FUNCTION_BLOCK ConvRobCtrl (* Basic Function Block Type *)
  (* Standard: 61499-2 *)
  (* Version 0.0, 5/12/2018, Aalto_IT, nxtControl GmbH, Template *)
  PACKAGE Main;
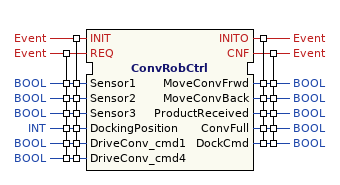
  EVENT_INPUT
    INIT WITH Sensor1, Sensor2, Sensor3, DockingPosition, DriveConv_cmd1, DriveConv_cmd4; (* Initialization Request *)
    REQ WITH Sensor1, Sensor2, Sensor3, DockingPosition, DriveConv_cmd1, DriveConv_cmd4; (* Normal Execution Request *)
  END_EVENT
  EVENT_OUTPUT
    INITO WITH MoveConvFrwd, MoveConvBack, ProductReceived, ConvFull, DockCmd; (* Initialization Confirm *)
    CNF WITH MoveConvFrwd, MoveConvBack, ProductReceived, ConvFull, DockCmd; (* Execution Confirmation *)
  END_EVENT
  VAR_INPUT
    Sensor1 : BOOL; (* Input event qualifier *)
    Sensor2 : BOOL;
    Sensor3 : BOOL;
    DockingPosition : INT;
    DriveConv_cmd1 : BOOL;
    DriveConv_cmd4 : BOOL;
  END_VAR
  VAR_OUTPUT
    MoveConvFrwd : BOOL; (* Output event qualifier *)
    MoveConvBack : BOOL;
    ProductReceived : BOOL;
    ConvFull : BOOL;
    DockCmd : BOOL;
  END_VAR
  VAR
    TimeStamp : DATE_AND_TIME;
  END_VAR
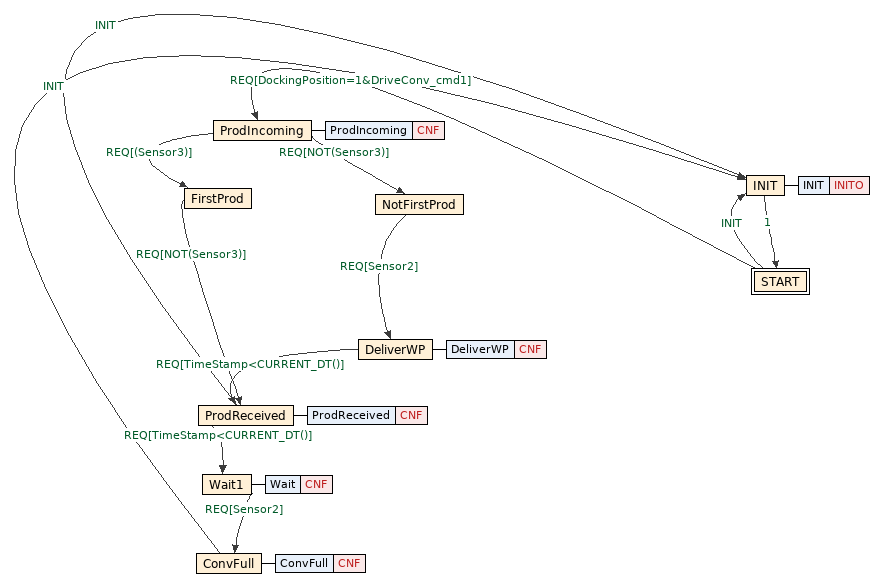
  EC_STATES
    START; (* Initial State *)
    INIT : INIT -> INITO; (* Initialization *)
    ProdIncoming : ProdIncoming -> CNF;
    FirstProd;
    NotFirstProd;
    DeliverWP : DeliverWP -> CNF;
    ConvFull : ConvFull -> CNF;
    ProdReceived : ProdReceived -> CNF;
    Wait1 : Wait -> CNF;
  END_STATES
  EC_TRANSITIONS
    START TO INIT := INIT;
    INIT TO START := 1;
    START TO ProdIncoming := REQ[DockingPosition=1&DriveConv_cmd1];
    ProdIncoming TO FirstProd := REQ[(Sensor3)];
    ProdIncoming TO NotFirstProd := REQ[NOT(Sensor3)];
    NotFirstProd TO DeliverWP := REQ[Sensor2];
    FirstProd TO ProdReceived := REQ[NOT(Sensor3)];
    ProdReceived TO INIT := INIT;
    DeliverWP TO ProdReceived := REQ[TimeStamp<CURRENT_DT()];
    Wait1 TO ConvFull := REQ[Sensor2];
    ConvFull TO INIT := INIT;
    ProdReceived TO Wait1 := REQ[TimeStamp<CURRENT_DT()];
  END_TRANSITIONS
  ALGORITHM INIT IN ST: (* Initialization algorithm *)
;
MoveConvBack := FALSE;
MoveConvFrwd := FALSE;
ConvFull := FALSE;
ProductReceived := FALSE;
DockCmd  := FALSE;
  END_ALGORITHM
  ALGORITHM REQ IN ST: (* Normally executed algorithm *)
;
  END_ALGORITHM
  ALGORITHM ProdIncoming IN ST:
;
// Drive Conveyor Inwards when always at Pos=1
MoveConvFrwd := FALSE;
MoveConvBack := TRUE;
ConvFull := FALSE;
ProductReceived := FALSE;
DockCmd  := FALSE;
  END_ALGORITHM
  ALGORITHM DeliverWP IN ST:
;
// use timer to deliver product once S2 is High.
TimeStamp := ADD_DT_TIME(CURRENT_DT(),T#2.5s);
MoveConvFrwd := FALSE;
MoveConvBack := TRUE;
ProductReceived := FALSE;
DockCmd  := FALSE;
  END_ALGORITHM
  ALGORITHM ConvFull IN ST:
;
MoveConvFrwd := FALSE;
MoveConvBack := FALSE;
//ProductReceived := TRUE;
ConvFull := TRUE;
DockCmd  := TRUE;
  END_ALGORITHM
  ALGORITHM FirstProd IN ST:
;
  END_ALGORITHM
  ALGORITHM ProdReceived IN ST:
;
MoveConvFrwd := FALSE;
MoveConvBack := FALSE;
ProductReceived := TRUE;
ConvFull := FALSE;
DockCmd  := FALSE;
TimeStamp := ADD_DT_TIME(CURRENT_DT(),T#1.0s);
  END_ALGORITHM
  ALGORITHM DriveConv IN ST:
;
MoveConvBack := FALSE;
MoveConvFrwd := FALSE;
ConvFull := FALSE;
ProductReceived := FALSE;
DockCmd  := FALSE;
  END_ALGORITHM
  ALGORITHM Wait IN ST:
;
MoveConvFrwd := FALSE;
MoveConvBack := FALSE;
ProductReceived := FALSE;
ConvFull := FALSE;
DockCmd  := FALSE;
  END_ALGORITHM
END_FUNCTION_BLOCK
